PROGRAM prg_PotentioMeter
VAR
	nPotentioMeter		AT		%I*		:INT;
	
	nPotPower			AT		%Q*		:INT := 32767; //Potentiometer voeden met 5V
	nWaarde				AT		%Q*		:REAL;
END_VAR

nWaarde := INT_TO_REAL(nPotentioMeter)*100 / 32767;

//Ander Oplossing:
//nWaarde:= INT_TO_REAL(nPotentioMeter) /327.67;

END_PROGRAM

(* stored: Version 1.1.0.1, ProductVersion 3.1.4024.15
   POU prg_PotentioMeter: Id {3e99a89c-11db-41cc-9b1c-93b47ac9ccc3}, SpecialFunc None *)
